// TIA Portal V17 export
// export: Created 2024-06-14T09:53:12.016692Z, ExportSetting WithDefaults, DisplayName Totally Integrated Automation Portal, DisplayVersion V17, DisplayName TIA Portal Openness, DisplayVersion V17, DisplayName TIA Portal Version Control Interface, DisplayVersion V17, DisplayName Simotion SCOUT TIA, DisplayVersion 5.4.3.0, DisplayName SINAMICS Startdrive Advanced, DisplayVersion V17 SP1 Update 1, DisplayName SINAMICS Startdrive G110M, G120, G120C, G120D, G120P, G115D, DisplayVersion V17 SP1 Update 1, DisplayName SINAMICS Startdrive G130, G150, S120, S150, SINAMICS MV, S210, DisplayVersion V17 SP1 Update 1, DisplayName STEP 7 Professional, DisplayVersion V17, DisplayName STEP 7 Safety, DisplayVersion V17, DisplayName WinCC Professional, DisplayVersion V17
FUNCTION "CORRECTION_SCALE" : Void   // FC4, LAD
{ S7_Optimized_Access := 'TRUE' }
VERSION : 0.1
// stored: AutoNumber false, IsIECCheckEnabled false, SetENOAutomatically false, UDAEnableTagReadback false
   VAR_TEMP
      cycle_start : Bool;
   END_VAR
BEGIN

REGION Network 1
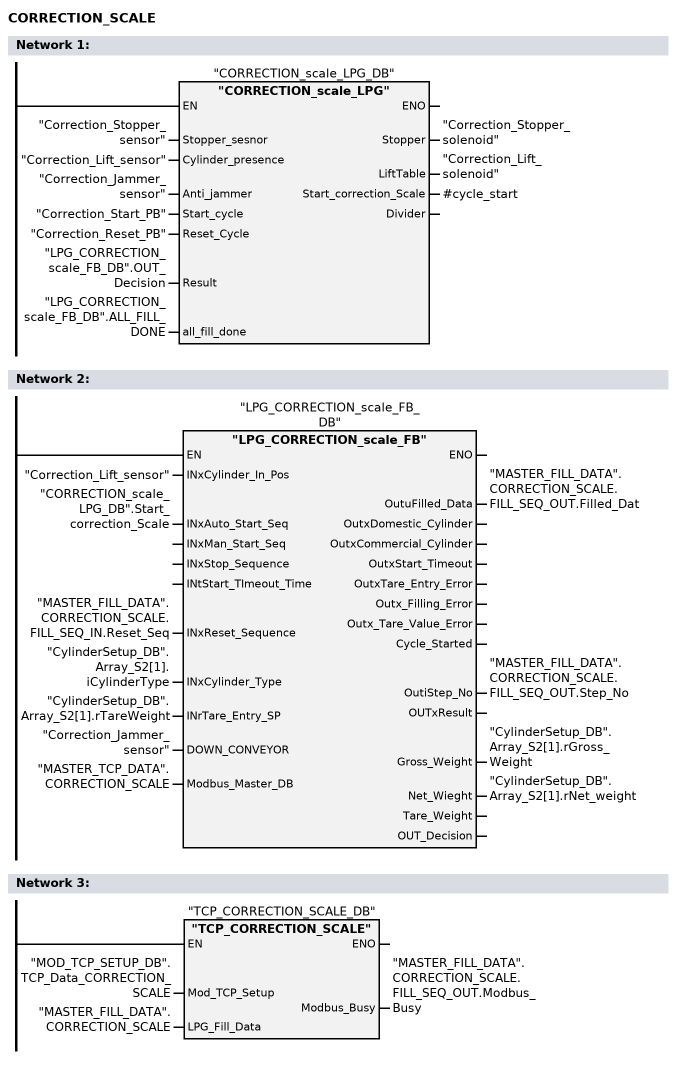
   RUNG wire#powerrail
      "CORRECTION_scale_LPG_DB"(Stopper_sesnor := "Correction_Stopper_sensor", Cylinder_presence := "Correction_Lift_sensor", Anti_jammer := "Correction_Jammer_sensor", Start_cycle := "Correction_Start_PB", Reset_Cycle := "Correction_Reset_PB", Result := "LPG_CORRECTION_scale_FB_DB".OUT_Decision, all_fill_done := "LPG_CORRECTION_scale_FB_DB".ALL_FILL_DONE, Stopper => "Correction_Stopper_solenoid", LiftTable => "Correction_Lift_solenoid", Start_correction_Scale => #cycle_start, Divider =>)
   END_RUNG
   // the same network as SCL:
   "CORRECTION_scale_LPG_DB"(Stopper_sesnor := "Correction_Stopper_sensor",   // "CORRECTION_scale_LPG"
                           Cylinder_presence := "Correction_Lift_sensor",
                           Anti_jammer := "Correction_Jammer_sensor",
                           Start_cycle := "Correction_Start_PB",
                           Reset_Cycle := "Correction_Reset_PB",
                           Result := "LPG_CORRECTION_scale_FB_DB".OUT_Decision,
                           all_fill_done := "LPG_CORRECTION_scale_FB_DB".ALL_FILL_DONE,
                           Stopper => "Correction_Stopper_solenoid",
                           LiftTable => "Correction_Lift_solenoid",
                           Start_correction_Scale => #cycle_start);
END_REGION

REGION Network 2
   RUNG wire#powerrail
      "LPG_CORRECTION_scale_FB_DB"(INxCylinder_In_Pos := "Correction_Lift_sensor", INxAuto_Start_Seq := "CORRECTION_scale_LPG_DB".Start_correction_Scale, INxMan_Start_Seq :=, INxStop_Sequence :=, INtStart_TImeout_Time :=, INxReset_Sequence := "MASTER_FILL_DATA".CORRECTION_SCALE.FILL_SEQ_IN.Reset_Seq, INxCylinder_Type := "CylinderSetup_DB".Array_S2[1].iCylinderType, INrTare_Entry_SP := "CylinderSetup_DB".Array_S2[1].rTareWeight, DOWN_CONVEYOR := "Correction_Jammer_sensor", Modbus_Master_DB := "MASTER_TCP_DATA".CORRECTION_SCALE, OutuFilled_Data => "MASTER_FILL_DATA".CORRECTION_SCALE.FILL_SEQ_OUT.Filled_Dat, OutxDomestic_Cylinder =>, OutxCommercial_Cylinder =>, OutxStart_Timeout =>, OutxTare_Entry_Error =>, Outx_Filling_Error =>, Outx_Tare_Value_Error =>, Cycle_Started =>, OutiStep_No => "MASTER_FILL_DATA".CORRECTION_SCALE.FILL_SEQ_OUT.Step_No, OUTxResult =>, Gross_Weight => "CylinderSetup_DB".Array_S2[1].rGross_Weight, Net_Wieght => "CylinderSetup_DB".Array_S2[1].rNet_weight, Tare_Weight =>, OUT_Decision =>)
   END_RUNG
   // the same network as SCL:
   "LPG_CORRECTION_scale_FB_DB"(INxCylinder_In_Pos := "Correction_Lift_sensor",   // "LPG_CORRECTION_scale_FB"
                           INxAuto_Start_Seq := "CORRECTION_scale_LPG_DB".Start_correction_Scale,
                           INxReset_Sequence := "MASTER_FILL_DATA".CORRECTION_SCALE.FILL_SEQ_IN.Reset_Seq,
                           INxCylinder_Type := "CylinderSetup_DB".Array_S2[1].iCylinderType,
                           INrTare_Entry_SP := "CylinderSetup_DB".Array_S2[1].rTareWeight,
                           DOWN_CONVEYOR := "Correction_Jammer_sensor",
                           Modbus_Master_DB := "MASTER_TCP_DATA".CORRECTION_SCALE,
                           OutuFilled_Data => "MASTER_FILL_DATA".CORRECTION_SCALE.FILL_SEQ_OUT.Filled_Dat,
                           OutiStep_No => "MASTER_FILL_DATA".CORRECTION_SCALE.FILL_SEQ_OUT.Step_No,
                           Gross_Weight => "CylinderSetup_DB".Array_S2[1].rGross_Weight,
                           Net_Wieght => "CylinderSetup_DB".Array_S2[1].rNet_weight);
END_REGION

REGION Network 3
   RUNG wire#powerrail
      "TCP_CORRECTION_SCALE_DB"(Mod_TCP_Setup := "MOD_TCP_SETUP_DB".TCP_Data_CORRECTION_SCALE, LPG_Fill_Data := "MASTER_FILL_DATA".CORRECTION_SCALE, Modbus_Busy => "MASTER_FILL_DATA".CORRECTION_SCALE.FILL_SEQ_OUT.Modbus_Busy)
   END_RUNG
   // the same network as SCL:
   "TCP_CORRECTION_SCALE_DB"(Mod_TCP_Setup := "MOD_TCP_SETUP_DB".TCP_Data_CORRECTION_SCALE,   // "TCP_CORRECTION_SCALE"
                           LPG_Fill_Data := "MASTER_FILL_DATA".CORRECTION_SCALE,
                           Modbus_Busy => "MASTER_FILL_DATA".CORRECTION_SCALE.FILL_SEQ_OUT.Modbus_Busy);
END_REGION
END_FUNCTION
